// TIA Portal V16 export
// export: Created 2021-11-12T13:31:05.291739Z, ExportSetting WithDefaults, DisplayName Totally Integrated Automation Portal, DisplayVersion V16 Update 3, DisplayName TIA Portal Version Control Interface, DisplayVersion V16 Update 2, DisplayName TIA Portal Openness, DisplayVersion V16 Update 3, DisplayName SINAMICS Startdrive Advanced, DisplayVersion V16 Update 5, DisplayName SINAMICS Startdrive G130, G150, S120, S150, SINAMICS MV, S210, DisplayVersion V16 Update 5, DisplayName SINAMICS Startdrive G110M, G120, G120C, G120D, G120P, G115D, DisplayVersion V16 Update 5, DisplayName STEP 7 Professional, DisplayVersion V16 Update 3, DisplayName STEP 7 Safety, DisplayVersion V16, DisplayName WinCC UA Professional, DisplayVersion V16 Update 3
DATA_BLOCK "DataCollInterface"   // DB46
{ S7_Optimized_Access := 'TRUE'; DB_Accessible_From_OPC_UA := 'FALSE' }
VERSION : 0.1
// stored: AutoNumber true, DBAccessibleFromOPCUA false, IsOnlyStoredInLoadMemory false, IsRetainMemResEnabled false, IsWriteProtectedInAS false, MemoryReserve 100
   VAR RETAIN
      DummyItem : "UDT_DataColl_Item";   // Dummy structure for Item
      DummyPeriodically : "UDT_DataColl_Periodically";   // Dummy structure for data archived periodically
      Item1 : "UDT_DataColl_Item";   // Item data to archive data block
      Item2 : "UDT_DataColl_Item";   // Item data to archive data block
      Periodically : "UDT_DataColl_Periodically";   // Periodically data to archive data block
   END_VAR
BEGIN
END_DATA_BLOCK
